TYPE SmokeControlParametersBase :
STRUCT
	SmokeControl: SmokeControlParameters;
END_STRUCT
END_TYPE

(* stored: Version 1.1.0.1, ProductVersion 3.1.4024.6
   DUT SmokeControlParametersBase: Id {31e8144e-1420-42f1-adcb-fd3ec93a9ef6} *)
